{attribute 'linkalways'} 
{attribute 'no_explicit_call' := 'This FB is a CLASS and must be accessed using methods or properties'}
{attribute 'enable_dynamic_creation'}
FUNCTION_BLOCK _FLOAT EXTENDS AliasDatatypeBase
VAR
	localData : FLOAT;
	activeData : REFERENCE TO FLOAT REF= localData;
	aliasBaseDatatype : _LREAL(localData);
END_VAR

PROPERTY PUBLIC Address : PVOID
GET
Address := ADR(activeData);
END_GET
END_PROPERTY

METHOD PUBLIC ClearReference
VAR_INPUT
END_VAR
activeData REF= localData;
SetBaseDatatypeReference();
END_METHOD

METHOD PUBLIC Clone : I_Datatype
VAR
    pClone : POINTER TO _FLOAT;
END_VAR
pClone := __NEW(_FLOAT(InitialValue := Value));
Clone := pClone^;
END_METHOD

METHOD FB_init : BOOL
VAR_INPUT
	bInitRetains : BOOL; // if TRUE, the retain variables are initialized (warm start / cold start)
	bInCopyCode : BOOL;  // if TRUE, the instance afterwards gets moved into the copy code (online change)
	InitialValue : FLOAT;
END_VAR
localData := InitialValue;
SetBaseDatatypeReference();
AddBaseDatatype(aliasBaseDatatype);
END_METHOD

PROPERTY PUBLIC Identifier : T_MAXSTRING
GET
Identifier := 'FLOAT';
END_GET
END_PROPERTY

METHOD PUBLIC MakeReferenceTo
VAR_INPUT
	ReferenceTarget : REFERENCE TO FLOAT;
END_VAR
activeData REF= ReferenceTarget;
SetBaseDatatypeReference();
END_METHOD

METHOD PROTECTED SetBaseDatatypeReference
VAR_INPUT
END_VAR
aliasBaseDatatype.MakeReferenceTo(activeData);
END_METHOD

PROPERTY PUBLIC Size : UDINT
GET
Size := SIZEOF(activeData);
END_GET
END_PROPERTY

METHOD TryMakeReferenceTo : BOOL
VAR_INPUT
	Target : I_Datatype;
END_VAR
VAR
	targetAsAlias : I_AliasDatatype;
	pTargetData : POINTER TO FLOAT;
END_VAR
IF NOT Target.TryResolveAsAliasDatatype(targetAsAlias) THEN
	RETURN;
END_IF

IF targetAsAlias.Identifier <> Identifier THEN
	RETURN;
END_IF

pTargetData := Target.Address;
activeData REF= pTargetData^;
SetBaseDatatypeReference();
TryMakeReferenceTo := TRUE;
END_METHOD

PROPERTY PUBLIC Value : REFERENCE TO FLOAT
GET
Value REF= activeData;
END_GET
END_PROPERTY

END_FUNCTION_BLOCK

(* stored: Version 1.1.0.1, ProductVersion 3.1.4024.12
   POU _FLOAT: Id {46f993eb-34f0-0567-1075-9e3d89c1ccc1}, SpecialFunc None
   Folder Constructor: Id {f89d074c-14a7-0fd5-0958-de635ff525e8}
   Folder Protected: Id {380a740d-c21e-081c-0279-bcad072a68fb}
   Property Address: Id {84ce47d2-ad6c-0425-3b46-0f0100f0fd03}
   Get Get: Id {bf795648-f9d4-0feb-0df2-982bc18fe192}
   Method ClearReference: Id {070a5628-5edf-0c2f-06e9-1ec2b80a9859}
   Method Clone: Id {1120d2ee-20fe-06f8-1143-dc604598fe10}
   Method FB_init: Id {2ffc75e4-47bc-0862-0cd8-d6b3dee6e1bc}
   Property Identifier: Id {af8147ed-4ebd-0b6d-2fe5-7b5b0da612e2}
   Get Get: Id {4e408498-fe2f-0ae9-0f49-faef22084d02}
   Method MakeReferenceTo: Id {54414441-95b9-0b3e-29df-75a3cefec034}
   Method SetBaseDatatypeReference: Id {e4414281-3d6b-09a5-3f96-499f36a9627b}
   Property Size: Id {23853b4d-332b-0164-3c7a-e1470276aae7}
   Get Get: Id {5e1bd266-3d38-02d8-04e1-731e18dbfc60}
   Method TryMakeReferenceTo: Id {df1e07a9-cce0-0954-2dcf-36c17d6a48a9}
   Property Value: Id {a60bd00b-30da-046f-3ab6-b29a83111a10}
   Get Get: Id {326fece7-0a78-04d4-366b-48ad3eadde7b} *)
